Fanuc KAREL source: kb00031.KL

-- PROVISIONAL review KL for V1013-1; original PC SHA256 c32b2fddc61bee2442b648215cc790208a906355c9794af1a1ebd9e21f3aca10
-- Incomplete behavior may be omitted. Consult companion uncertainty JSON. Do not deploy.
PROGRAM KB00031
%NOLOCKGROUP
BEGIN
  -- UNRESOLVED_PC offsets 5-16; opcodes 2E,23
  -- UNRESOLVED_PC offsets 21-30; opcodes 3F,75
  -- UNRESOLVED_PC offsets 35-42; opcodes 9D,23
  -- UNRESOLVED_PC offsets 47-71; opcodes 27,22,22,2A,22,31
  -- UNRESOLVED_PC offsets 76-80; opcodes 7F
END KB00031
